Staubli VAL3: chkDrivesSwOff.pgx

program chkDrivesSwOff()
  local bool l_bDrvSwOnDis
  local num l_i
begin
  // 检测驱动器“switch on disabled"的状态
  bDrivesSwOnDis=true
  for l_i=0 to nAxesSum-1
    bSWOnDis[l_i]=(diSwOnDis[l_i]==true)
    bDrivesSwOnDis=bDrivesSwOnDis and bSWOnDis[l_i]
  endFor
  //
end
